(* PLC project Unnamed, Unknown Unnamed 1 *)
(* stored: creationDateTime 2022-08-16T15:49:17, modificationDateTime 2025-10-23T11:18:57 *)

PROGRAM Blink
  VAR
    blink_led0 AT %QX0.0 : BOOL;
    blink_led1 AT %QX0.1 : BOOL;
    blink_led2 AT %QX0.2 : BOOL;
  END_VAR
  VAR
    TON0 : TON;
    TOF0 : TOF;
  END_VAR
  VAR
    timer_preset_ms AT %QW0 : INT := 500;
  END_VAR
  VAR
    timer_preset_t : TIME := T#500ms;
    MSCONV : REAL := 1000.0;
  END_VAR

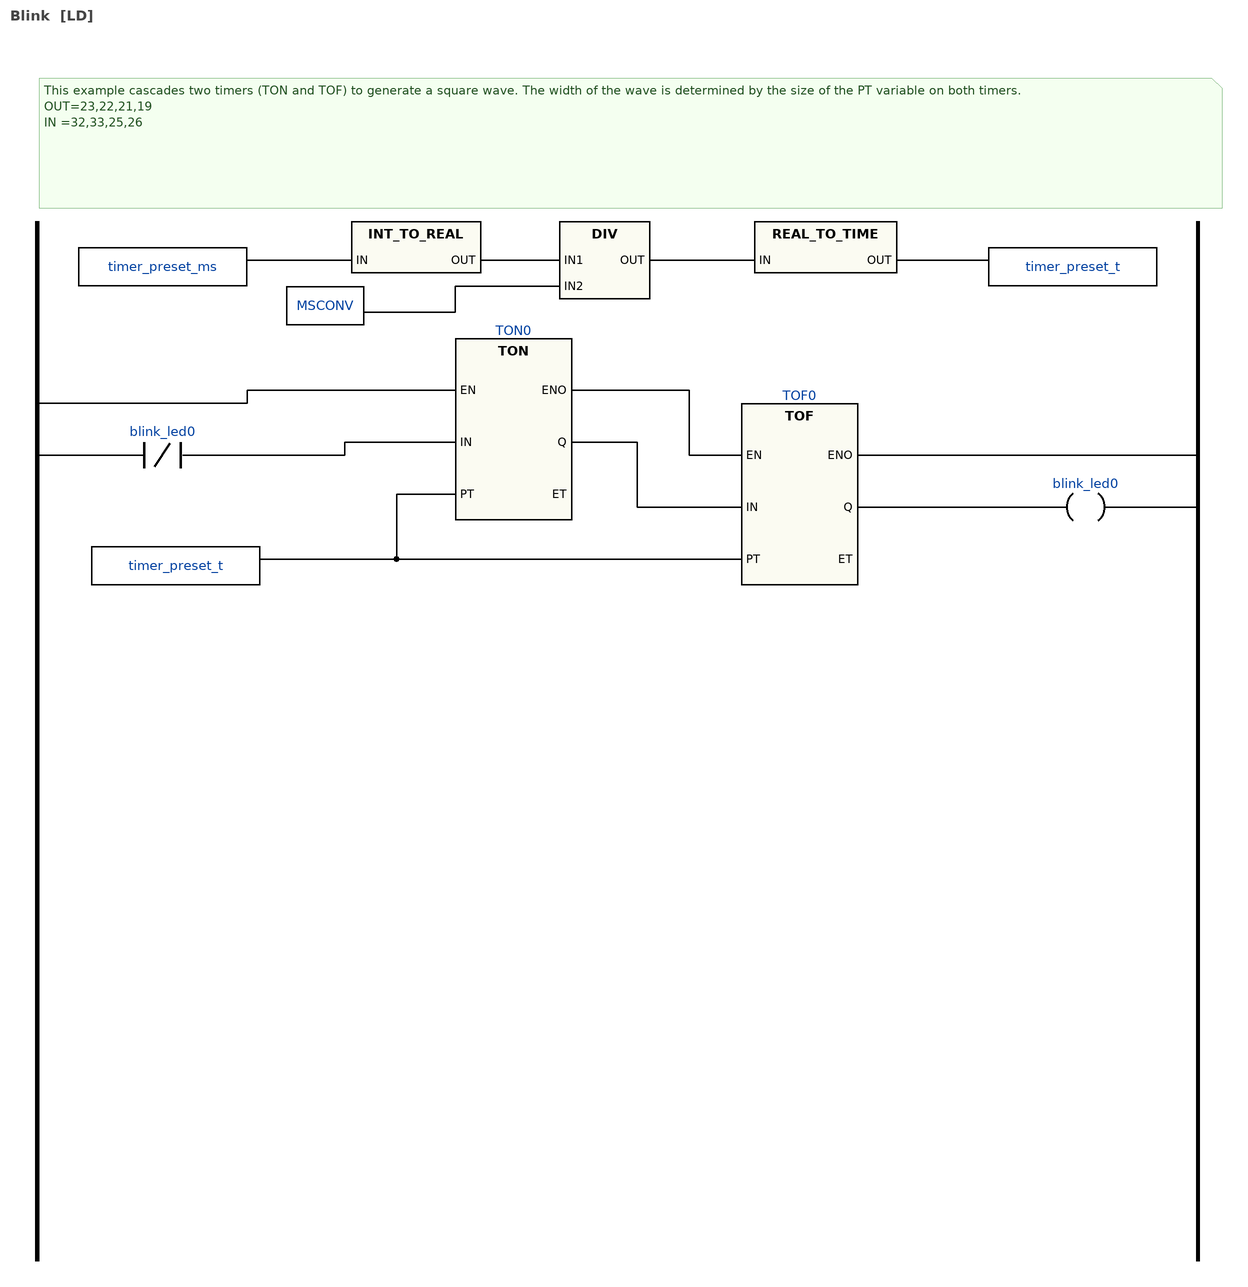
(* LD diagram, written out as Structured Text *)
(* This example cascades two timers (TON and TOF) to generate a square wave. The width of the wave is determined by the size of the PT variable on both timers.
OUT=23,22,21,19
IN =32,33,25,26 *)
TON0(IN := NOT blink_led0, PT := timer_preset_t);
TOF0(EN := TON0.ENO, IN := TON0.Q, PT := timer_preset_t);
blink_led0 := TOF0.Q;
timer_preset_t := REAL_TO_TIME(INT_TO_REAL(timer_preset_ms) / MSCONV);
END_PROGRAM

CONFIGURATION Config0
  RESOURCE Res0 ON PLC
    TASK task0(INTERVAL := T#20ms, PRIORITY := 0);
    PROGRAM instance0 WITH task0 : Blink;
  END_RESOURCE
END_CONFIGURATION
